TYPE E_MethodState :
(
	Ready := 0,
	Busy := 1,
	Error := 2 
)USINT;
END_TYPE

(* stored: Version 1.1.0.1, ProductVersion 3.1.0.25
   DUT E_MethodState: Id {419b5adf-007b-459e-b1fc-da811d64f048} *)
